INTERFACE I_Base extends __SYSTEM.IQueryInterface

METHOD M_Request : BOOL
VAR_INPUT
	eState:		E_Base;
END_VAR
END_METHOD

PROPERTY P_Logger : I_Logger
GET
END_GET
SET
END_SET
END_PROPERTY

PROPERTY PUBLIC P_State : E_Base
GET
END_GET
END_PROPERTY

END_INTERFACE

(* stored: Version 1.1.0.1
   Itf I_Base: Id {ada3f4ee-e52c-4b2e-ad47-2676c314edf3}
   Method M_Request: Id {0f1926ad-fb7a-0886-3826-aeef678c8655}
   Property P_Logger: Id {6fb3a8fe-2739-06e9-3894-49e798facdba}
   Get Get: Id {581d3e03-4c18-00d3-2756-8605376a3eb3}
   Set Set: Id {123d7bb0-a994-01b6-0a58-cdba6ee7e68b}
   Property P_State: Id {519f0641-a13c-0e6f-16fe-695b8f49bbd7}
   Get Get: Id {a6309e82-4735-0d58-29bd-fc8c104809a5} *)
